FUNCTION F_ITC_SendECR : BOOL
(**************************************************************************************
 * 	Application		:	BoxControl Framework
 *	Revision		:	$Revision: 404529 $
 *	Revision date	:	$Date: 2018-04-23 08:21:38 +0200 (Mo., 23 Apr 2018) $
 *	Last changed by	:	$Author: b7bolm $
 *	URL				:	$URL: http://almscdc.swisslog.com/repo/SWPD/Development/BoxControlFramework/20_Release/trunk/01_Software/BCF/BCF/JumpStart/20_Product/10_App/11_Com/10_Lib/10_Conv/11_ITC/F_ITC_SendECR.TcPOU $
 *
 *	Purpose			:	Wrap message - ECR
 *
 * ------------------------------------------------------------------------------------
 *	Copyright Swisslog [IP AG], Switzerland. All rights reserved.
 * 
 * ------------------------------------------------------------------------------------
 *	
 * 	Revision History: 
 *
 * 	VERSION			DATE			INITIALS			DESCRIPTION
 *	0.1				01.01.2001		swl					Example
 *
 **************************************************************************************)
VAR_INPUT
	eChannelSrc		: E_MFCS_Channel; // Source communicaton channel	
	ElementName		: STRING(Conveyor.POSITION_STRINGLENGTH); // The conveyor element which reports its status
	Code			: INT; // ControlCode
	Variable		: DINT; // Variable
	eReturnCode		: E_ErrorConv; // Return code
END_VAR
VAR
	ECR				: ST_ITC_ECR; 
END_VAR

// Map values
ECR.Position := ElementName;
ECR.Code := Code;
ECR.Variable := Variable;
ECR.ReturnCode := eReturnCode;

// Forward to ITC
F_ITC_SendECR := fbITC_Manager.M_SendData(
					meChannel	:= eChannelSrc,
					mMsgType	:= E_ITC_MsgTypeConv.ELEMENT_CONTROL_REPLY,
					mpData		:= ADR(ECR),
					mLen		:= SIZEOF(ECR));

END_FUNCTION

(* stored: Version 1.1.0.1, ProductVersion 3.1.4022.12
   POU F_ITC_SendECR: Id {3d34f0a4-33a8-4c17-bb36-42dcb1e2086e}, SpecialFunc None *)
